FUNCTION_BLOCK FB_MaterialService EXTENDS FB_ServiceBase
VAR_INPUT
END_VAR
VAR_OUTPUT
END_VAR
VAR
END_VAR

END_FUNCTION_BLOCK

(* stored: Version 1.1.0.1, ProductVersion 3.1.4026.18
   POU FB_MaterialService: Id {27a75cf1-edc2-4d2c-b790-ee82654cc92e}, SpecialFunc None *)
